INTERFACE I_RpcManagerConfig

PROPERTY PUBLIC ContentType_Json : T_MAXSTRING
GET
END_GET
END_PROPERTY

METHOD PUBLIC TryGetAcceptResponseFormatFromRequest : BOOL
VAR_INPUT
	Request : I_Request;
	Destination : ANY;
END_VAR
END_METHOD

METHOD PUBLIC TryGetContentTypeFromRequest : BOOL
VAR_INPUT
	Request : I_Request;
	Destination : ANY;
END_VAR
END_METHOD

METHOD PUBLIC TryGetMethodNameFromRequest : BOOL
VAR_INPUT
	Request : I_Request;
	Destination : ANY;
END_VAR
END_METHOD

METHOD PUBLIC TryGetTypeFromRequest : BOOL
VAR_INPUT
	Request : I_Request;
	Destination : ANY;
END_VAR
END_METHOD

END_INTERFACE

(* stored: Version 1.1.0.1, ProductVersion 3.1.4024.12
   Itf I_RpcManagerConfig: Id {4a4f0798-ed83-499b-b5a8-20a54d5c473a}
   Property ContentType_Json: Id {c2359f88-ebc0-4bc5-bd89-97e2615909d5}
   Get Get: Id {3d6b8bfc-8450-4f79-8aa0-01f67fb99dab}
   Method TryGetAcceptResponseFormatFromRequest: Id {e6b357e2-8223-477a-ab4e-7919087a405d}
   Method TryGetContentTypeFromRequest: Id {bfab91a5-16ef-465f-8d15-2a8d8c434dfc}
   Method TryGetMethodNameFromRequest: Id {5c2608d7-66af-4db9-bf73-ee9acebab690}
   Method TryGetTypeFromRequest: Id {fb413ab0-893d-4594-a530-fabc1706787a} *)
